PROGRAM MAIN
VAR
	bDoubleSquareScal, bAddVec, bCrossProd, bScaleVec: BOOL;
	eError : E_Error;
	fbScalar : FB_Scalar(2.2);
	fbVec1 : FB_Vector(1,2,3);
	fbVec2 : FB_Vector(3,2,1);
END_VAR

IF bDoubleSquareScal THEN 
	bDoubleSquareScal := FALSE;
	fbScalar.Times(fbScalar.Plus(fbScalar));
	END_IF

IF bAddVec THEN
	bAddVec := FALSE;
	fbVec1.Plus(fbVec2);
	END_IF
	
IF bCrossProd THEN
	bCrossProd := FALSE;
	fbVec1.Times(fbVec2);
	END_IF
	
IF bScaleVec THEN
	bScaleVec := FALSE;
	fbVec1.Times(fbScalar);
	END_IF

END_PROGRAM

(* stored: Version 1.1.0.1, ProductVersion 3.1.4024.4
   POU MAIN: Id {36d1238f-0d46-4dcc-84f8-262dc2254684}, SpecialFunc None *)
